// TIA Portal V18 export
TYPE "SubAssembly Check_ShW"
// stored: IsFailsafeCompliant false
   STRUCT
      Trigger : Bool;
      Result : Int;
      Completed : Bool;
      Q_ID : "SubAssemblyID_ShW";
   END_STRUCT;
END_TYPE
